TYPE WcStateBase_A2171C4E :
STRUCT
END_STRUCT
END_TYPE
